TYPE AX5000_P_0097 :
STRUCT
	Motor_brake_unlocked:BOOL;
	Rsvd:ARRAY[0..14] OF BOOL;
END_STRUCT
END_TYPE

(* stored: Version 1.1.0.1, ProductVersion 3.1.4024.16
   DUT AX5000_P_0097: Id {2b38a40a-fd98-422b-bdd7-746862b89d63} *)
